INTERFACE I_RecipeManagment EXTENDS I_Component

{attribute 'monitoring' := 'call'}
PROPERTY AutoLoadChangesToActive : BOOL
SET
END_SET
END_PROPERTY

{attribute 'monitoring' := 'call'}
PROPERTY ChangesPending : BOOL
GET
END_GET
END_PROPERTY

METHOD LoadChangesToActive
VAR_INPUT
END_VAR
END_METHOD

END_INTERFACE

(* stored: Version 1.1.0.1, ProductVersion 3.1.4026.18
   Itf I_RecipeManagment: Id {aba03838-8842-45de-a315-eb954587180b}
   Property AutoLoadChangesToActive: Id {2c157dc0-d485-43f8-af78-3fdecff89fd7}
   Set Set: Id {d83a91fb-e1f3-4641-ac72-d95566d2bc71}
   Property ChangesPending: Id {1d47bcf0-d076-4f47-b143-84642a87977b}
   Get Get: Id {fce04d95-e0f7-4d9d-a396-fee135bbcfe9}
   Method LoadChangesToActive: Id {f42c7b8c-41c9-4027-95f4-d77ffc93688e} *)
